{attribute 'linkalways'} 
{attribute 'no_explicit_call' := 'This FB is a CLASS and must be accessed using methods or properties'}
{attribute 'enable_dynamic_creation'}
FUNCTION_BLOCK _ETcVnDistanceTransformationMask EXTENDS EnumDatatypeBase
VAR
	localData : ETcVnDistanceTransformationMask;
	activeData : REFERENCE TO ETcVnDistanceTransformationMask;
	enumBaseDatatype : _DINT(localData);
END_VAR

METHOD PRIVATE AddLocalEnumeration
VAR_INPUT
	Enumeration : T_MAXSTRING;
	Value : ETcVnDistanceTransformationMask;
END_VAR
AddEnumeration(Enumeration, Value);
END_METHOD

PROPERTY PUBLIC Address : PVOID
GET
Address := ADR(activeData);
END_GET
END_PROPERTY

METHOD PUBLIC ClearReference
VAR_INPUT
END_VAR
activeData REF= localData;
SetBaseDatatypeReference();
END_METHOD

METHOD PUBLIC Clone : I_Datatype
VAR
    pClone : POINTER TO _ETcVnDistanceTransformationMask;
END_VAR
pClone := __NEW(_ETcVnDistanceTransformationMask(InitialValue := Value));
Clone := pClone^;
END_METHOD

METHOD FB_init : BOOL
VAR_INPUT
	bInitRetains : BOOL; // if TRUE, the retain variables are initialized (warm start / cold start)
	bInCopyCode : BOOL;  // if TRUE, the instance afterwards gets moved into the copy code (online change)
	InitialValue : ETcVnDistanceTransformationMask;
END_VAR
localData := InitialValue;
AddBaseDatatype(enumBaseDatatype);
ClearReference();

AddLocalEnumeration('TCVN_DTM_PRECISE', ETcVnDistanceTransformationMask.TCVN_DTM_PRECISE);
AddLocalEnumeration('TCVN_DTM_3', ETcVnDistanceTransformationMask.TCVN_DTM_3);
AddLocalEnumeration('TCVN_DTM_5', ETcVnDistanceTransformationMask.TCVN_DTM_5);
END_METHOD

PROPERTY PUBLIC Identifier : T_MAXSTRING
GET
Identifier := 'ETcVnDistanceTransformationMask';
END_GET
END_PROPERTY

METHOD IsEnumeratorValueEqual : BOOL
VAR_INPUT
	Enumerator : I_KeyValueForwardEnumerator;
END_VAR
VAR
	storedValue : ETcVnDistanceTransformationMask;
END_VAR
IF NOT Enumerator.TryGet(storedValue) THEN
	RETURN;
END_IF

IsEnumeratorValueEqual := storedValue = activeData;
END_METHOD

METHOD PUBLIC MakeReferenceTo
VAR_INPUT
	ReferenceTarget : REFERENCE TO ETcVnDistanceTransformationMask;
END_VAR
activeData REF= ReferenceTarget;
SetBaseDatatypeReference();
END_METHOD

METHOD PROTECTED SetBaseDatatypeReference
VAR_INPUT
END_VAR
enumBaseDatatype.MakeReferenceTo(activeData);
END_METHOD

PROPERTY PUBLIC Size : UDINT
GET
Size := SIZEOF(activeData);
END_GET
END_PROPERTY

METHOD TryMakeReferenceTo : BOOL
VAR_INPUT
	Target : I_Datatype;
END_VAR
VAR
	targetAsEnum : I_EnumDatatype;
	pTargetData : POINTER TO ETcVnDistanceTransformationMask;
END_VAR
IF NOT Target.TryResolveAsEnumDatatype(targetAsEnum) THEN
	RETURN;
END_IF

IF targetAsEnum.Identifier <> Identifier THEN
	RETURN;
END_IF

pTargetData := Target.Address;
activeData REF= pTargetData^;
SetBaseDatatypeReference();
TryMakeReferenceTo := TRUE;
END_METHOD

PROPERTY PUBLIC Value : ETcVnDistanceTransformationMask
GET
Value := activeData;
END_GET
SET
activeData := Value;
END_SET
END_PROPERTY

END_FUNCTION_BLOCK

(* stored: Version 1.1.0.1, ProductVersion 3.1.4024.12
   POU _ETcVnDistanceTransformationMask: Id {d6e72ada-7ce2-4439-9a1d-7ada40770705}, SpecialFunc None
   Folder Constructor: Id {520a5628-f7d1-45ec-baba-00688797585d}
   Folder Private: Id {0a74f357-efd3-416f-a145-0735a96b8d1d}
   Folder Protected: Id {3b046f0c-f9c5-4f68-894a-e4d6f36aa041}
   Method AddLocalEnumeration: Id {49ea389f-d464-4cb0-a4ac-36dacde4f97d}
   Property Address: Id {d26001c6-ec0e-407d-850e-64b23ec63c12}
   Get Get: Id {c1385c1f-7716-476a-9fd6-65fadbdf54cb}
   Method ClearReference: Id {8c989dcd-173f-4d6e-9081-d82db24ba41a}
   Method Clone: Id {3ab8f42d-9b01-4d01-9b5a-0f07b0a16c00}
   Method FB_init: Id {2cca96ec-f573-4cec-9b1f-258bec251b3d}
   Property Identifier: Id {ff89f445-b554-4937-abf7-78f745904705}
   Get Get: Id {b7fb5806-c0aa-4024-a29e-47bf88c808a0}
   Method IsEnumeratorValueEqual: Id {d088e5e2-e98e-479f-befc-c206b1a78929}
   Method MakeReferenceTo: Id {063280d2-33b5-4b6b-b053-da245cab307c}
   Method SetBaseDatatypeReference: Id {77507094-cd4f-4ca8-9d49-45df8132cee7}
   Property Size: Id {e2e60b9e-4528-4912-96a3-95d74d006c64}
   Get Get: Id {440039ee-ff34-4666-9f57-0f5bd675e3bd}
   Method TryMakeReferenceTo: Id {dd741a17-045e-43f9-8ab5-e4bf72d437e6}
   Property Value: Id {8a220ac2-40cf-4d05-8368-fe68938753e1}
   Get Get: Id {87264889-a985-4f23-8934-f45a384387e1}
   Set Set: Id {20bae960-66b3-483d-a856-27158e202e1b} *)
